FUNCTION_BLOCK Test_GetTestHandlesEmptyList EXTENDS T_UnitTestBase IMPLEMENTS I_UnitTest
VAR
    List : T_ListOfTests(Capacity := 10);
END_VAR

METHOD Init
List.Clear();
END_METHOD

METHOD RunTest
VAR_OUTPUT
    TestCompleted : BOOL;
    TestFailed    : BOOL;
END_VAR
VAR_INST
    TestNumber2 : I_UnitTest;
END_VAR
TestNumber2 := List.GetTest(2);

AssertTrue(Source    := TestName,
             Condition := (TestNumber2 = 0),
             Message   := 'Interface pointer TestNumber2 was not zero',
             Failed    => TestFailed);

TestCompleted := TRUE;
END_METHOD

END_FUNCTION_BLOCK

(* stored: Version 1.1.0.1, ProductVersion 3.1.4024.12
   POU Test_GetTestHandlesEmptyList: Id {0377225d-b398-4c13-bbd5-f5d116644514}, SpecialFunc None
   Method Init: Id {f5a8aaee-52fb-4db1-98b0-740d059321f3}
   Method RunTest: Id {c6dfbf80-c24b-481a-868f-5d5f6bcb529b} *)
